Universal Robots PolyScope program: xmlrpc_example_listadinamica.urp

Program xmlrpc_example (installation=default directory=/home/ur/ursim-current/programs createdIn=5.16.1 lastSavedIn=5.16.1 robotSerialNumber=20195299999)
Calibrated DH parameters: a=[0, -0.6127, -0.57155, 0, 0, 0]; d=[0.1807, 0, 0, 0.17415, 0.11985, 0.11655]; alpha=[1.570796, 0, 0, 1.570796, -1.570796, 0]; deltaTheta=[0, 0, 0, 0, 0, 0]
InitVariablesNode
BeforeStart
  camera := rpc_factory("xmlrpc","https:10.0.2.20")
Robot Program (runOnlyOnce=false)
  Loop While (checkContinuously=false) expression=True
    next_pose := camera.get_pose()
    If next_pose[0]==0
      Popup Warning (haltProgram=false message=No hay  mas posiciones a las que moverse inputType=Text)
    MoveJ speed 60 deg/s, acceleration 80 deg/s^2 (useActiveTCP=true) feature=Base
      Waypoint Variable (Variable): variable=next_pose
